FUNCTION_BLOCK NullError_TestSuite EXTENDS TcUnit.FB_TestSuite

TestErrorType();
TestMessage();

METHOD PUBLIC TestErrorType
VAR
	error : NullError;
END_VAR
TEST('TestErrorType');

AssertEquals_String(
	Actual := error.ErrorType,
	Expected := '',
	Message := 'Did not return the expected ErrorType'
);

TEST_FINISHED();
END_METHOD

METHOD PUBLIC TestMessage
VAR
	error : NullError;
END_VAR
TEST('TestMessage');

AssertEquals_String(
	Actual := error.Message,
	Expected := '',
	Message := 'Did not return the expected Message'
);

TEST_FINISHED();
END_METHOD

END_FUNCTION_BLOCK

(* stored: Version 1.1.0.1, ProductVersion 3.1.4024.12
   POU NullError_TestSuite: Id {1b850d10-5b07-4fc3-9e5b-bb907eb1956c}, SpecialFunc None
   Method TestErrorType: Id {641a95c2-206b-4d79-bdfd-51f5226ec6a1}
   Method TestMessage: Id {dd6f8769-f16f-4d91-9c79-6fd4795285ab} *)
